(* CoDeSys 2.3.9.50 project: inicio.pr6 *)
(* Libraries: STANDARD.LB6 5.6.98 12:03:02 *)

(* Global variable list: TwinCAT_Import *)
VAR_GLOBAL (* DO NOT CHANGE THIS SHEET MANUALLY! *)
	PlcInVar_0	AT %QB128:	USINT;
	PlcInVar_1	AT %QB129:	USINT;
	PlcInVar_2	AT %QB130:	USINT;
	PlcInVar_3	AT %QB131:	USINT;
	PlcInVar_4	AT %QB132:	USINT;
	PlcInVar_5	AT %QB133:	USINT;
	PlcInVar_6	AT %QB134:	USINT;
	PlcInVar_7	AT %QB135:	USINT;
	PlcInVar_8	AT %QB136:	USINT;
	PlcInVar_9	AT %QB137:	USINT;
	PlcInVar_10	AT %QB138:	USINT;
	PlcInVar_11	AT %QB139:	USINT;
	PlcInVar_12	AT %QB140:	USINT;
	PlcInVar_13	AT %QB141:	USINT;
	PlcInVar_14	AT %QB142:	USINT;
	PlcInVar_15	AT %QB143:	USINT;
	PlcOutVar_0	AT %IB128:	USINT;
	PlcOutVar_1	AT %IB129:	USINT;
	PlcOutVar_2	AT %IB130:	USINT;
	PlcOutVar_3	AT %IB131:	USINT;
	PlcOutVar_4	AT %IB132:	USINT;
	PlcOutVar_5	AT %IB133:	USINT;
	PlcOutVar_6	AT %IB134:	USINT;
	PlcOutVar_7	AT %IB135:	USINT;
	PlcOutVar_8	AT %IB136:	USINT;
	PlcOutVar_9	AT %IB137:	USINT;
	PlcOutVar_10	AT %IB138:	USINT;
	PlcOutVar_11	AT %IB139:	USINT;
	PlcOutVar_12	AT %IB140:	USINT;
	PlcOutVar_13	AT %IB141:	USINT;
	PlcOutVar_14	AT %IB142:	USINT;
	PlcOutVar_15	AT %IB143:	USINT;

	Terminal_2_KL1408_1_Input	AT %IX0.0:	BOOL; (* YL-01 (WATER DEFENSE) *)
	Terminal_2_KL1408_2_Input	AT %IX0.1:	BOOL; (* YL-02 (RECOVERY TANK LOW LEVEL) *)
Terminal_2_KL1408_3_Input	AT %IX0.2:	BOOL; (* YL-03 (RECOVERY TANK HIGH LEVEL) *)
Terminal_2_KL1408_4_Input	AT %IX0.3:	BOOL; (* YL-04 (RECOVERY TANK HIGH/HIGH LEVEL) *)
Terminal_2_KL1408_5_Input	AT %IX0.4:	BOOL; (* YL-05 (STATIC REEL A) *)
Terminal_2_KL1408_6_Input	AT %IX0.5:	BOOL; (* YL-06 (HYDRANT COUPLER) *)
Terminal_2_KL1408_7_Input	AT %IX0.6:	BOOL; (* YL-07 (PLATFORM POSITION) *)
	Terminal_2_KL1408_8_Input	AT %IX0.7:	BOOL; (* YL-08 (FRONT STABILIZER UP) *)

	Terminal_3_KL1408_1_Input	AT %IX1.0:	BOOL; (* YL-09 (SIDE STABILIZER UP) *)
Terminal_3_KL1408_2_Input	AT %IX1.1:	BOOL; (* YL-10 (FRONT STABILIZER DOWN) *)
Terminal_3_KL1408_3_Input	AT %IX1.2:	BOOL; (* YL-11 (LOCK INLET EXTENSION) *)
	Terminal_3_KL1408_4_Input	AT %IX1.3:	BOOL; (* YL-12 (UNDERWING SIDE NOZZLE) *)
Terminal_3_KL1408_5_Input	AT %IX1.4:	BOOL; 
	Terminal_3_KL1408_6_Input	AT %IX1.5:	BOOL;
Terminal_3_KL1408_7_Input	AT %IX1.6:	BOOL; (* YL-15 (+15 SIGNAL) *)
	Terminal_3_KL1408_8_Input	AT %IX1.7:	BOOL; (* YL-16 (PLATFORM DOOR LOCK) *)

Terminal_4_KL1408_1_Input	AT %IX2.0:	BOOL; (* YL-17 (UNDERWING PLATFORM NOZZLE A) *)
Terminal_4_KL1408_2_Input	AT %IX2.1:	BOOL; (* YL-18 (UNDERWING PLATFORM NOZZLE B) *)
Terminal_4_KL1408_3_Input	AT %IX2.2:	BOOL; (* YL-19 (LASER PLATFORM SWITCH) *)
Terminal_4_KL1408_4_Input	AT %IX2.3:	BOOL; (* YL-20 (PANEL & VISUAL SAMPLER LIGHT SWITCH) *)
Terminal_4_KL1408_5_Input	AT %IX2.4:	BOOL; (* YL-21 (INTERLOCK OVERRIDE) *)
Terminal_4_KL1408_6_Input	AT %IX2.5:	BOOL; (* YL-22 (AUTO START/STOP ENGINE SWITCH) *)
Terminal_4_KL1408_7_Input	AT %IX2.6:	BOOL; (* YL-23 (EFSO) *)
Terminal_4_KL1408_8_Input	AT %IX2.7:	BOOL; (* YL-24 (REWIND HOSE REEL SWITCH) *)

	Terminal_5_KL1408_1_Input	AT %IX3.0:	BOOL; (* YL-53 (UNDERWING NOZZLE PLATFORM CAP A) *)
	Terminal_5_KL1408_2_Input	AT %IX3.1:	BOOL;
Terminal_5_KL1408_3_Input	AT %IX3.2:	BOOL; (* YL-27 (START BARTEC) *)
Terminal_5_KL1408_4_Input	AT %IX3.3:	BOOL; (* YL-28 (DP STOP) *)
	Terminal_5_KL1408_5_Input	AT %IX3.4:	BOOL; (* YL-29 (AFGUARD 15 PPM) *)
Terminal_5_KL1408_6_Input	AT %IX3.5:	BOOL; (* YL-30 (AFGUARD 30 PPM) *)
Terminal_5_KL1408_7_Input	AT %IX3.6:	BOOL; (* YL-31 (AIR PRESSURE) *)
Terminal_5_KL1408_8_Input	AT %IX3.7:	BOOL; (* YL-32 (STABILIZERS UP SWITCH) *)

Terminal_6_KL1408_1_Input	AT %IX4.0:	BOOL; (* YL-33 (STABILIZERS DOWN SWITCH) *)
	Terminal_6_KL1408_2_Input	AT %IX4.1:	BOOL; (* YL-34 (DEADMAN OVERRIDE SWITCH) *)
Terminal_6_KL1408_3_Input	AT %IX4.2:	BOOL; (* YL-35 (RECOVERY TANK SWITCH) *)
Terminal_6_KL1408_4_Input	AT %IX4.3:	BOOL; (* YL-36 (WORK LIGHT SWITCH) *)
Terminal_6_KL1408_5_Input	AT %IX4.4:	BOOL; (* YL-37 (ULTRASONIC LEFT PLATFORM SENSOR) *)
Terminal_6_KL1408_6_Input	AT %IX4.5:	BOOL; (* YL-38 (ULTRASONIC RIGHT PLATFORM SENSOR) *)
Terminal_6_KL1408_7_Input	AT %IX4.6:	BOOL; (* YL-39 (PLATFORM UP SWITCH) *)
Terminal_6_KL1408_8_Input	AT %IX4.7:	BOOL; (* YL-40 (PLATFORM DOWN SWITCH) *)

Terminal_7_KL1408_1_Input	AT %IX5.0:	BOOL; (* YL-41 (LIMIT PLATFORM SWITCH) *)
Terminal_7_KL1408_2_Input	AT %IX5.1:	BOOL; (* YL-42 (DEADMAN HANDLE INTERLOCK) *)
Terminal_7_KL1408_3_Input	AT %IX5.2:	BOOL; (* YL-43 (DEADMAN HANDLE ACTIVE) *)
Terminal_7_KL1408_4_Input	AT %IX5.3:	BOOL; (* YL-44 (DEADMAN LIGHT TIMER) *)
Terminal_7_KL1408_5_Input	AT %IX5.4:	BOOL; (* YL-51 (STATIC REEL B) *)
Terminal_7_KL1408_6_Input	AT %IX5.5:	BOOL; (* YL-52 (DRIVER SIDE DOOR) *)
Terminal_7_KL1408_7_Input	AT %IX5.6:	BOOL; 
Terminal_7_KL1408_8_Input	AT %IX5.7:	BOOL; 

Terminal_8_KL1408_1_Input	AT %IX6.0:	BOOL; (* YL-45 (EXTRA CAB INPUT SIGNAL) *)
Terminal_8_KL1408_2_Input	AT %IX6.1:	BOOL; 
Terminal_8_KL1408_3_Input	AT %IX6.2:	BOOL; (* YL-47 (HANDBRAKE ACTIVE) *)
Terminal_8_KL1408_4_Input	AT %IX6.3:	BOOL; (* YL-48 (PTO ACTIVE) *)
Terminal_8_KL1408_5_Input	AT %IX6.4:	BOOL; (* YL-49 (SPEED 5 km/h) *)
	Terminal_8_KL1408_6_Input	AT %IX6.5:	BOOL; (* YL-50 (ENGINE RUNNING +D SIGNAL) *)
Terminal_8_KL1408_7_Input	AT %IX6.6:	BOOL; 
Terminal_8_KL1408_8_Input	AT %IX6.7:	BOOL; 


	Terminal_9_KL2424_1_Output	AT %QX0.0:	BOOL;
	Terminal_9_KL2424_2_Output	AT %QX0.1:	BOOL;
	Terminal_9_KL2424_3_Output	AT %QX0.2:	BOOL;
	Terminal_9_KL2424_4_Output	AT %QX0.3:	BOOL;

	Terminal_10_KL2424_1_Output	AT %QX0.4:	BOOL;
	Terminal_10_KL2424_2_Output	AT %QX0.5:	BOOL;
	Terminal_10_KL2424_3_Output	AT %QX0.6:	BOOL;
	Terminal_10_KL2424_4_Output	AT %QX0.7:	BOOL;

	Terminal_11_KL2424_1_Output	AT %QX1.0:	BOOL;
	Terminal_11_KL2424_2_Output	AT %QX1.1:	BOOL;
	Terminal_11_KL2424_3_Output	AT %QX1.2:	BOOL;
	Terminal_11_KL2424_4_Output	AT %QX1.3:	BOOL;

	Terminal_12_KL2408_1_Output	AT %QX1.4:	BOOL;
	Terminal_12_KL2408_2_Output	AT %QX1.5:	BOOL;
	Terminal_12_KL2408_3_Output	AT %QX1.6:	BOOL;
	Terminal_12_KL2408_4_Output	AT %QX1.7:	BOOL;
	Terminal_12_KL2408_5_Output	AT %QX2.0:	BOOL;
	Terminal_12_KL2408_6_Output	AT %QX2.1:	BOOL;
	Terminal_12_KL2408_7_Output	AT %QX2.2:	BOOL;
	Terminal_12_KL2408_8_Output	AT %QX2.3:	BOOL;

	Terminal_13_KL2408_1_Output	AT %QX2.4:	BOOL;
	Terminal_13_KL2408_2_Output	AT %QX2.5:	BOOL;
	Terminal_13_KL2408_3_Output	AT %QX2.6:	BOOL;
	Terminal_13_KL2408_4_Output	AT %QX2.7:	BOOL;
	Terminal_13_KL2408_5_Output	AT %QX3.0:	BOOL;
	Terminal_13_KL2408_6_Output	AT %QX3.1:	BOOL;
	Terminal_13_KL2408_7_Output	AT %QX3.2:	BOOL;
	Terminal_13_KL2408_8_Output	AT %QX3.3:	BOOL;

	Terminal_14_KL2408_1_Output	AT %QX3.4:	BOOL;
	Terminal_14_KL2408_2_Output	AT %QX3.5:	BOOL;
	Terminal_14_KL2408_3_Output	AT %QX3.6:	BOOL;
	Terminal_14_KL2408_4_Output	AT %QX3.7:	BOOL;
	Terminal_14_KL2408_5_Output	AT %QX4.0:	BOOL;
	Terminal_14_KL2408_6_Output	AT %QX4.1:	BOOL;
	Terminal_14_KL2408_7_Output	AT %QX4.2:	BOOL;
         Terminal_14_KL2408_8_Output	AT %QX4.3:	BOOL;

	Terminal_15_KL2408_1_Output	AT %QX4.4:	BOOL;
	Terminal_15_KL2408_2_Output	AT %QX4.5:	BOOL;
	Terminal_15_KL2408_3_Output	AT %QX4.6:	BOOL;(* YL-50 (INTERLOCK LIGHT) *)
	Terminal_15_KL2408_4_Output	AT %QX4.7:	BOOL;
	Terminal_15_KL2408_5_Output	AT %QX5.0:	BOOL;
	Terminal_15_KL2408_6_Output	AT %QX5.1:	BOOL;
	Terminal_15_KL2408_7_Output	AT %QX5.2:	BOOL;
	Terminal_15_KL2408_8_Output	AT %QX5.3:	BOOL;
END_VAR

(* POU MAIN, LD *)
PROGRAM MAIN
VAR

END_VAR
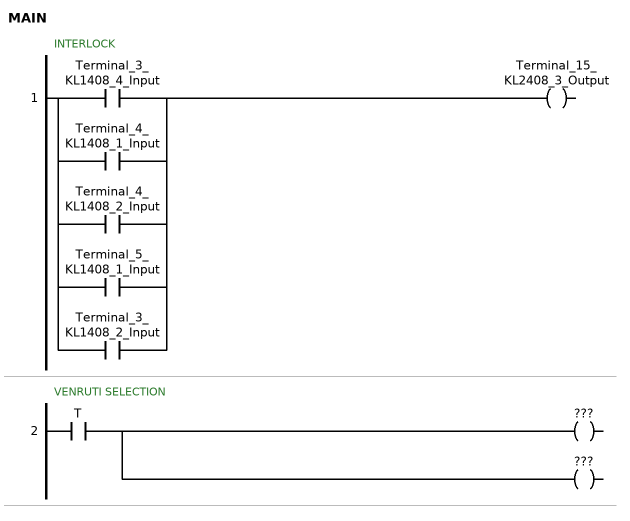
_LD_ (* Ladder Diagram *)
NETWORK 1 (* INTERLOCK *)
	{ [Terminal_3_KL1408_4_Input] | [Terminal_4_KL1408_1_Input] | [Terminal_4_KL1408_2_Input] | [Terminal_5_KL1408_1_Input] | [Terminal_3_KL1408_2_Input] } --- (Terminal_15_KL2408_3_Output)
NETWORK 2 (* VENRUTI SELECTION *)
	[T] --- (???) (???)
_END_LD_
(* the same logic as Structured Text *)
(* Network 1 *)
Terminal_15_KL2408_3_Output := Terminal_3_KL1408_4_Input OR Terminal_4_KL1408_1_Input OR Terminal_4_KL1408_2_Input OR Terminal_5_KL1408_1_Input OR Terminal_3_KL1408_2_Input;
(* Network 2: see the listing above *)
END_PROGRAM
